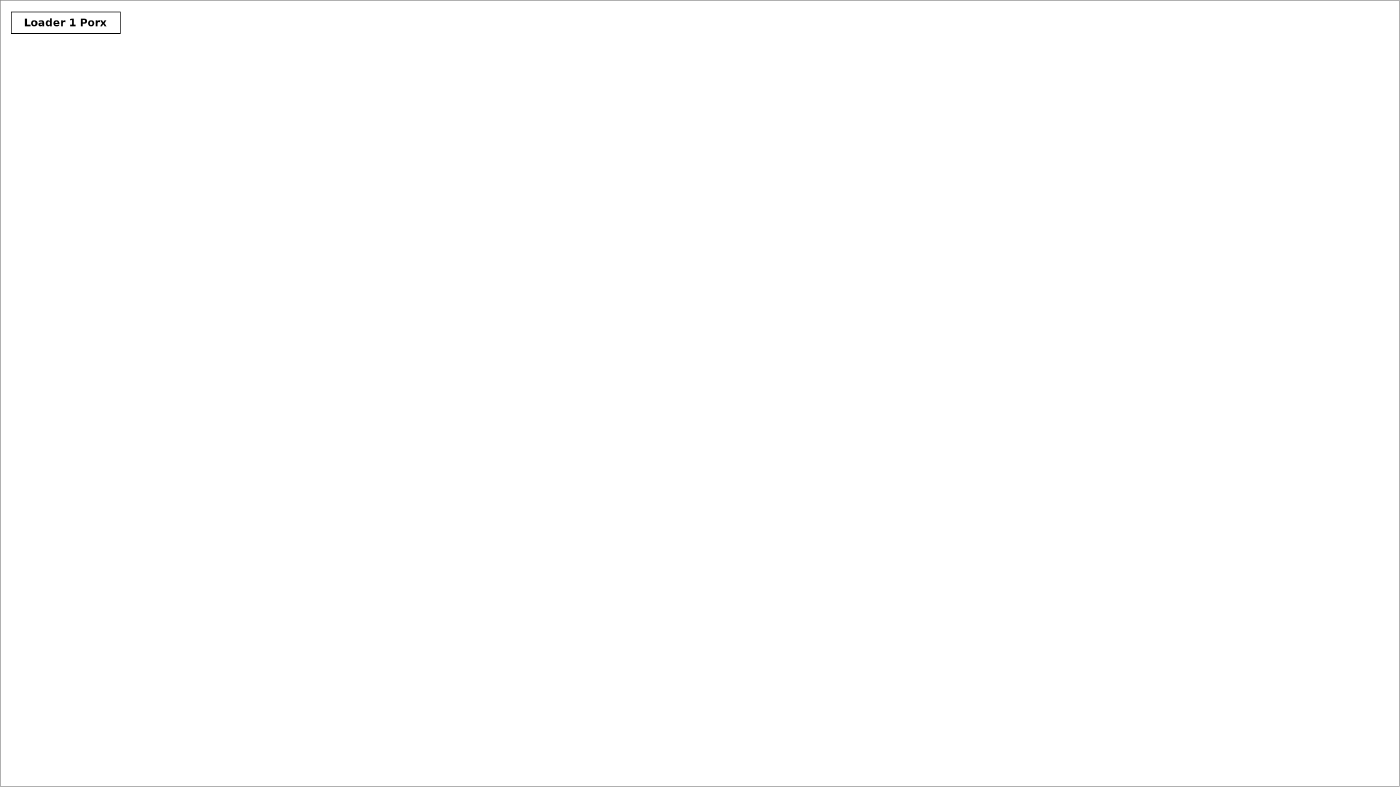
VISUALIZATION Main_Page  // 1920x1080
    RoundedRectangle (15,16 150x30), "Loader 1 Porx", tooltip "Connected to IN1-3", colour toggle: Loaders.Loader_1.Level_Prox
END_VISUALIZATION

(* stored: Version 1.1.0.1, ProductVersion 3.1.4024.13
   Visu Main_Page: Id {6c8f2165-dd8b-43ff-8820-3d7ebdc658fd} *)
